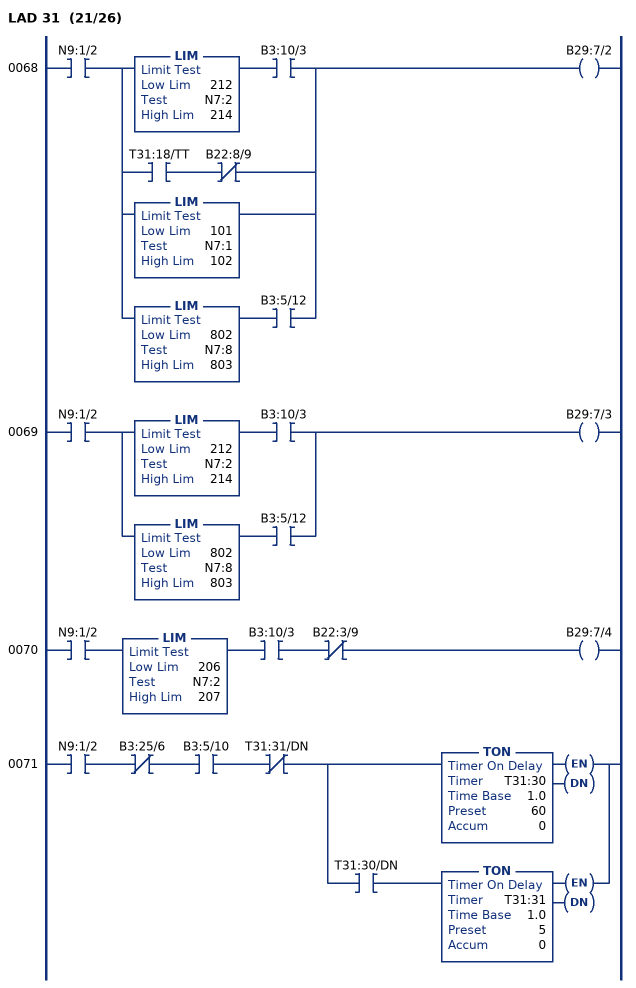
% Rung: 68 %
SOR XIC N9:1/2 BST LIM 212 N7:2 214 XIC B3:10/3 NXB XIC T31:18/TT XIO B22:8/9 NXB LIM 101 N7:1 102 NXB LIM 802 N7:8 803 XIC B3:5/12 BND OTE B29:7/2 EOR
% Rung: 69 %
SOR XIC N9:1/2 BST LIM 212 N7:2 214 XIC B3:10/3 NXB LIM 802 N7:8 803 XIC B3:5/12 BND OTE B29:7/3 EOR
% Rung: 70 %
SOR XIC N9:1/2 LIM 206 N7:2 207 XIC B3:10/3 XIO B22:3/9 OTE B29:7/4 EOR
% Rung: 71 %
SOR XIC N9:1/2 XIO B3:25/6 XIC B3:5/10 XIO T31:31/DN BST TON T31:30 1.0 60 0 NXB XIC T31:30/DN TON T31:31 1.0 5 0 BND EOR

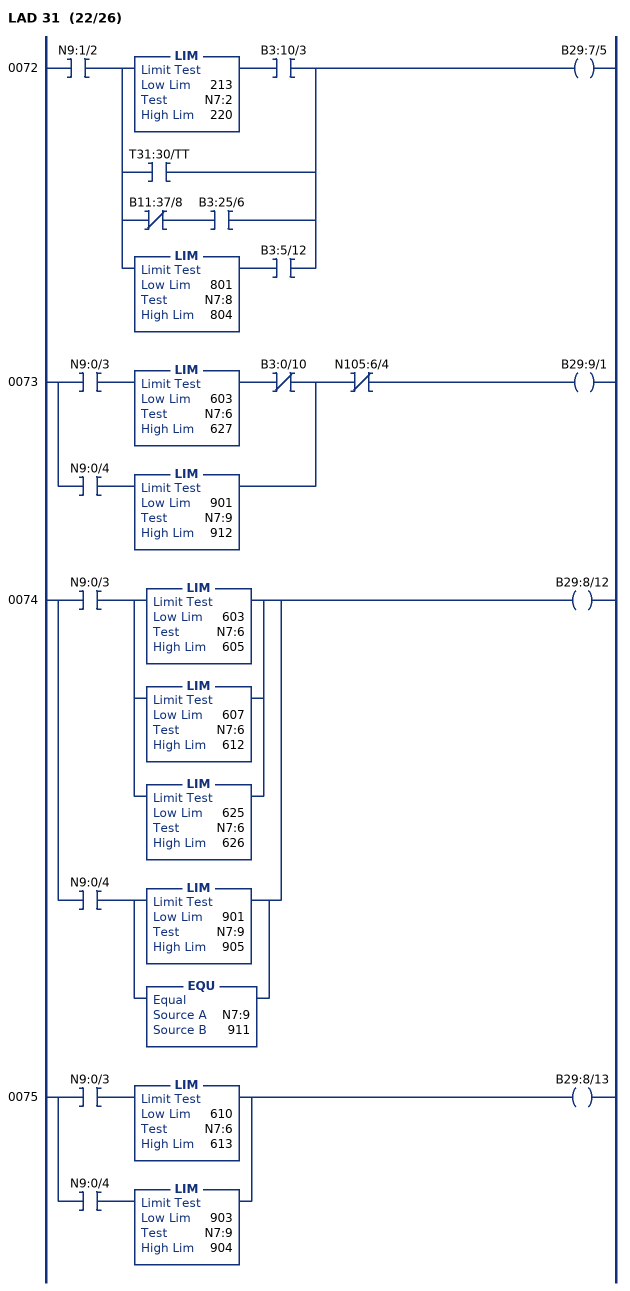
% Rung: 72 %
SOR XIC N9:1/2 BST LIM 213 N7:2 220 XIC B3:10/3 NXB XIC T31:30/TT NXB XIO B11:37/8 XIC B3:25/6 NXB LIM 801 N7:8 804 XIC B3:5/12 BND OTE B29:7/5 EOR
% Rung: 73 %
SOR BST XIC N9:0/3 LIM 603 N7:6 627 XIO B3:0/10 NXB XIC N9:0/4 LIM 901 N7:9 912 BND XIO N105:6/4 OTE B29:9/1 EOR
% Rung: 74 %
SOR BST XIC N9:0/3 BST LIM 603 N7:6 605 NXB LIM 607 N7:6 612 NXB LIM 625 N7:6 626 BND NXB XIC N9:0/4 BST LIM 901 N7:9 905 NXB EQU N7:9 911 BND BND OTE B29:8/12 EOR
% Rung: 75 %
SOR BST XIC N9:0/3 LIM 610 N7:6 613 NXB XIC N9:0/4 LIM 903 N7:9 904 BND OTE B29:8/13 EOR

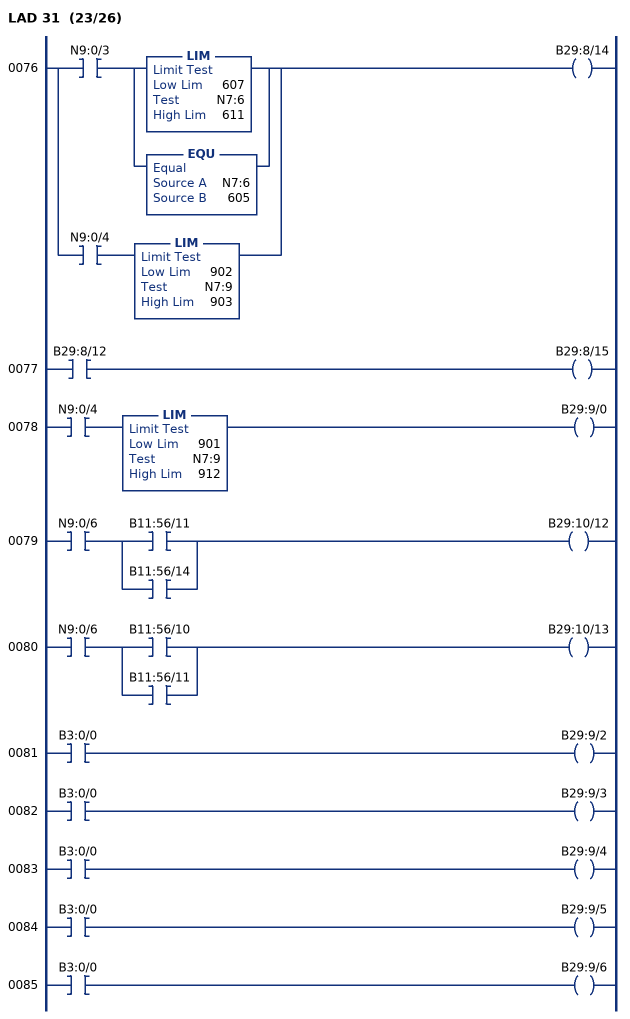
% Rung: 76 %
SOR BST XIC N9:0/3 BST LIM 607 N7:6 611 NXB EQU N7:6 605 BND NXB XIC N9:0/4 LIM 902 N7:9 903 BND OTE B29:8/14 EOR
% Rung: 77 %
SOR XIC B29:8/12 OTE B29:8/15 EOR
% Rung: 78 %
SOR XIC N9:0/4 LIM 901 N7:9 912 OTE B29:9/0 EOR
% Rung: 79 %
SOR XIC N9:0/6 BST XIC B11:56/11 NXB XIC B11:56/14 BND OTE B29:10/12 EOR
% Rung: 80 %
SOR XIC N9:0/6 BST XIC B11:56/10 NXB XIC B11:56/11 BND OTE B29:10/13 EOR
% Rung: 81 %
SOR XIC B3:0/0 OTE B29:9/2 EOR
% Rung: 82 %
SOR XIC B3:0/0 OTE B29:9/3 EOR
% Rung: 83 %
SOR XIC B3:0/0 OTE B29:9/4 EOR
% Rung: 84 %
SOR XIC B3:0/0 OTE B29:9/5 EOR
% Rung: 85 %
SOR XIC B3:0/0 OTE B29:9/6 EOR

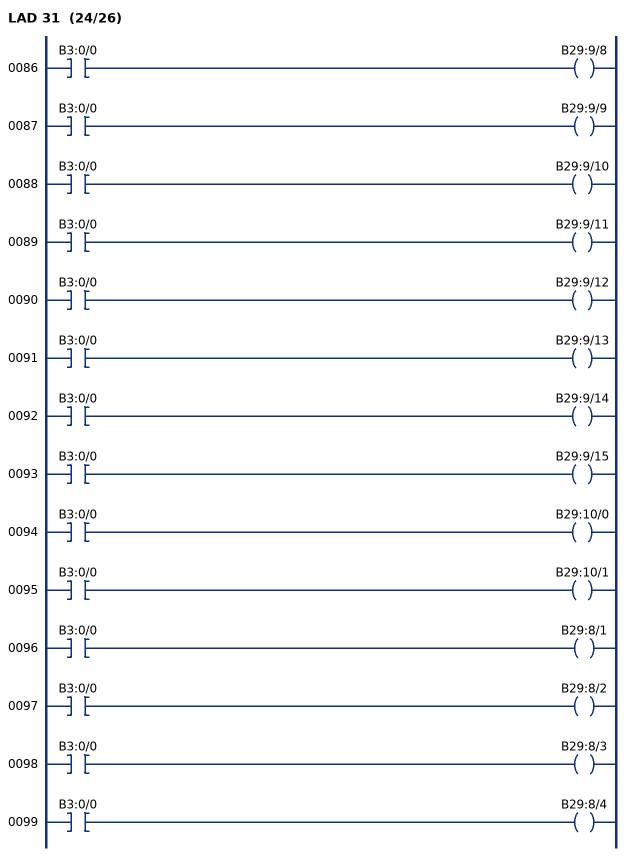
% Rung: 86 %
SOR XIC B3:0/0 OTE B29:9/8 EOR
% Rung: 87 %
SOR XIC B3:0/0 OTE B29:9/9 EOR
% Rung: 88 %
SOR XIC B3:0/0 OTE B29:9/10 EOR
% Rung: 89 %
SOR XIC B3:0/0 OTE B29:9/11 EOR
% Rung: 90 %
SOR XIC B3:0/0 OTE B29:9/12 EOR
% Rung: 91 %
SOR XIC B3:0/0 OTE B29:9/13 EOR
% Rung: 92 %
SOR XIC B3:0/0 OTE B29:9/14 EOR
% Rung: 93 %
SOR XIC B3:0/0 OTE B29:9/15 EOR
% Rung: 94 %
SOR XIC B3:0/0 OTE B29:10/0 EOR
% Rung: 95 %
SOR XIC B3:0/0 OTE B29:10/1 EOR
% Rung: 96 %
SOR XIC B3:0/0 OTE B29:8/1 EOR
% Rung: 97 %
SOR XIC B3:0/0 OTE B29:8/2 EOR
% Rung: 98 %
SOR XIC B3:0/0 OTE B29:8/3 EOR
% Rung: 99 %
SOR XIC B3:0/0 OTE B29:8/4 EOR

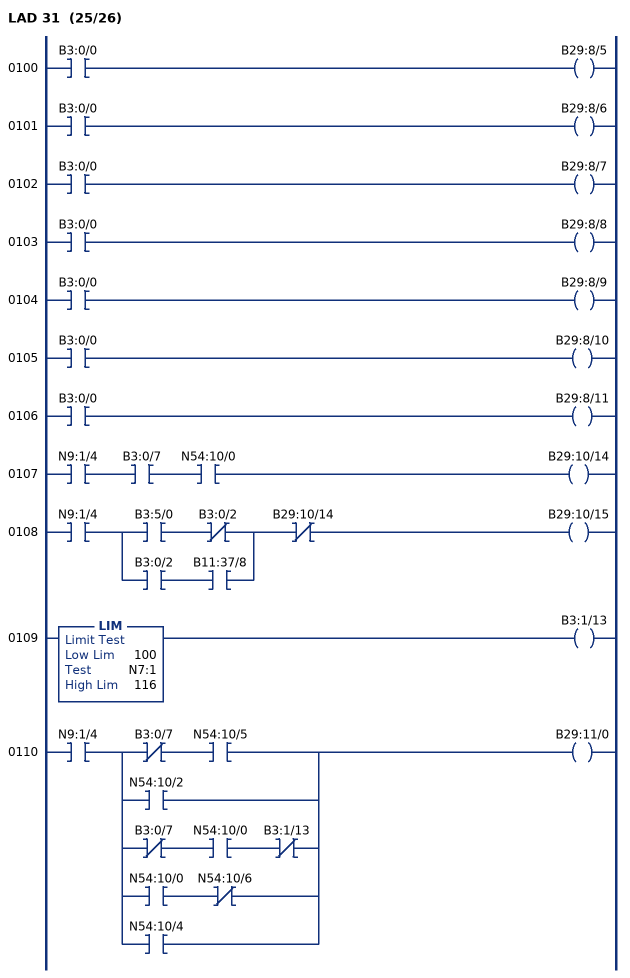
% Rung: 100 %
SOR XIC B3:0/0 OTE B29:8/5 EOR
% Rung: 101 %
SOR XIC B3:0/0 OTE B29:8/6 EOR
% Rung: 102 %
SOR XIC B3:0/0 OTE B29:8/7 EOR
% Rung: 103 %
SOR XIC B3:0/0 OTE B29:8/8 EOR
% Rung: 104 %
SOR XIC B3:0/0 OTE B29:8/9 EOR
% Rung: 105 %
SOR XIC B3:0/0 OTE B29:8/10 EOR
% Rung: 106 %
SOR XIC B3:0/0 OTE B29:8/11 EOR
% Rung: 107 %
SOR XIC N9:1/4 XIC B3:0/7 XIC N54:10/0 OTE B29:10/14 EOR
% Rung: 108 %
SOR XIC N9:1/4 BST XIC B3:5/0 XIO B3:0/2 NXB XIC B3:0/2 XIC B11:37/8 BND XIO B29:10/14 OTE B29:10/15 EOR
% Rung: 109 %
SOR LIM 100 N7:1 116 OTE B3:1/13 EOR
% Rung: 110 %
SOR XIC N9:1/4 BST XIO B3:0/7 XIC N54:10/5 NXB XIC N54:10/2 NXB XIO B3:0/7 XIC N54:10/0 XIO B3:1/13 NXB XIC N54:10/0 XIO N54:10/6 NXB XIC N54:10/4 BND OTE B29:11/0 EOR

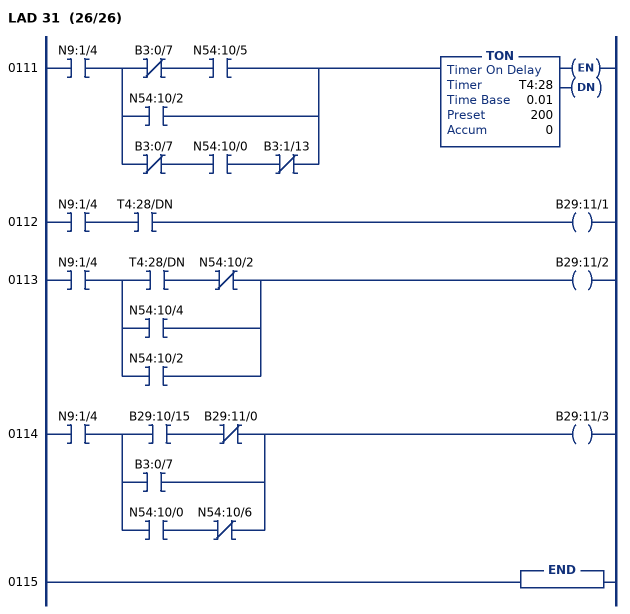
% Rung: 111 %
SOR XIC N9:1/4 BST XIO B3:0/7 XIC N54:10/5 NXB XIC N54:10/2 NXB XIO B3:0/7 XIC N54:10/0 XIO B3:1/13 BND TON T4:28 0.01 200 0 EOR
% Rung: 112 %
SOR XIC N9:1/4 XIC T4:28/DN OTE B29:11/1 EOR
% Rung: 113 %
SOR XIC N9:1/4 BST XIC T4:28/DN XIO N54:10/2 NXB XIC N54:10/4 NXB XIC N54:10/2 BND OTE B29:11/2 EOR
% Rung: 114 %
SOR XIC N9:1/4 BST XIC B29:10/15 XIO B29:11/0 NXB XIC B3:0/7 NXB XIC N54:10/0 XIO N54:10/6 BND OTE B29:11/3 EOR
% Rung: 115 %
SOR END EOR

LADDER 32
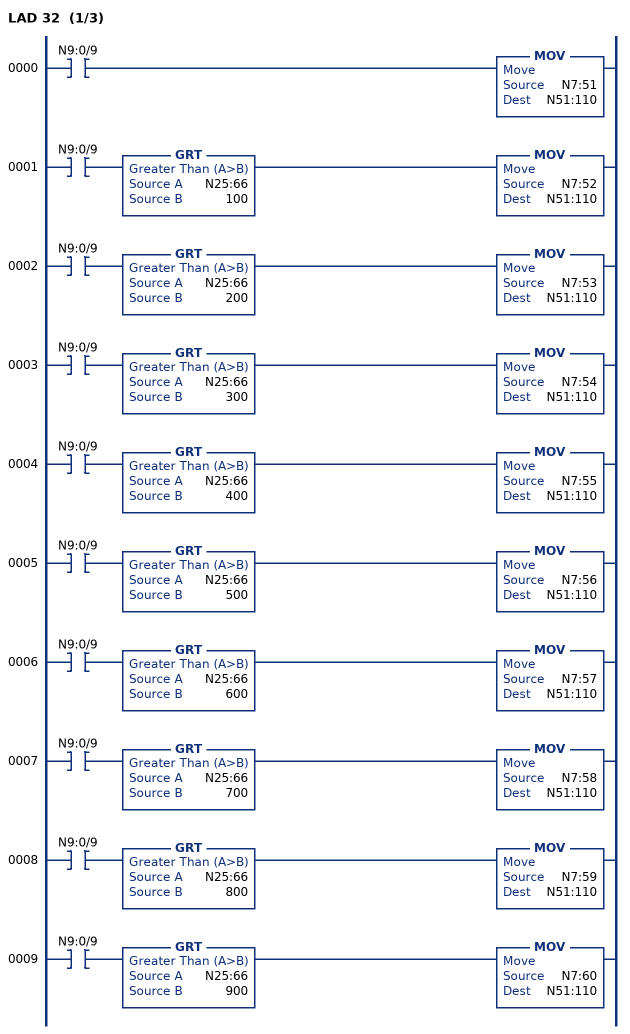
% Rung: 0 %
SOR XIC N9:0/9 MOV N7:51 N51:110 EOR
% Rung: 1 %
SOR XIC N9:0/9 GRT N25:66 100 MOV N7:52 N51:110 EOR
% Rung: 2 %
SOR XIC N9:0/9 GRT N25:66 200 MOV N7:53 N51:110 EOR
% Rung: 3 %
SOR XIC N9:0/9 GRT N25:66 300 MOV N7:54 N51:110 EOR
% Rung: 4 %
SOR XIC N9:0/9 GRT N25:66 400 MOV N7:55 N51:110 EOR
% Rung: 5 %
SOR XIC N9:0/9 GRT N25:66 500 MOV N7:56 N51:110 EOR
% Rung: 6 %
SOR XIC N9:0/9 GRT N25:66 600 MOV N7:57 N51:110 EOR
% Rung: 7 %
SOR XIC N9:0/9 GRT N25:66 700 MOV N7:58 N51:110 EOR
% Rung: 8 %
SOR XIC N9:0/9 GRT N25:66 800 MOV N7:59 N51:110 EOR
% Rung: 9 %
SOR XIC N9:0/9 GRT N25:66 900 MOV N7:60 N51:110 EOR

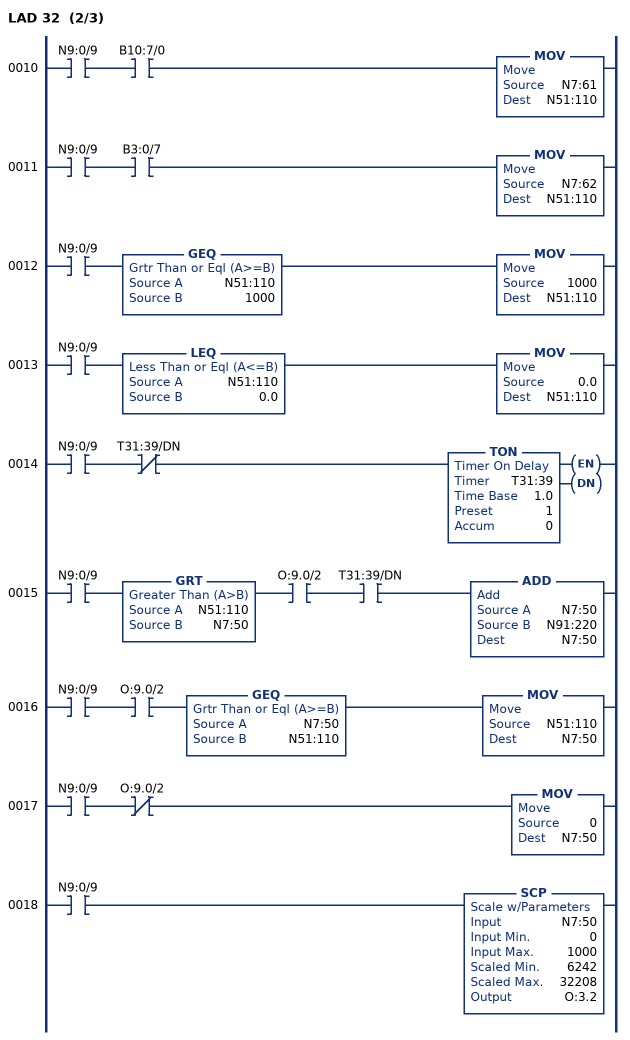
% Rung: 10 %
SOR XIC N9:0/9 XIC B10:7/0 MOV N7:61 N51:110 EOR
% Rung: 11 %
SOR XIC N9:0/9 XIC B3:0/7 MOV N7:62 N51:110 EOR
% Rung: 12 %
SOR XIC N9:0/9 GEQ N51:110 1000 MOV 1000 N51:110 EOR
% Rung: 13 %
SOR XIC N9:0/9 LEQ N51:110 0.0 MOV 0.0 N51:110 EOR
% Rung: 14 %
SOR XIC N9:0/9 XIO T31:39/DN TON T31:39 1.0 1 0 EOR
% Rung: 15 %
SOR XIC N9:0/9 GRT N51:110 N7:50 XIC O:9.0/2 XIC T31:39/DN ADD N7:50 N91:220 N7:50 EOR
% Rung: 16 %
SOR XIC N9:0/9 XIC O:9.0/2 GEQ N7:50 N51:110 MOV N51:110 N7:50 EOR
% Rung: 17 %
SOR XIC N9:0/9 XIO O:9.0/2 MOV 0 N7:50 EOR
% Rung: 18 %
SOR XIC N9:0/9 SCP N7:50 0 1000 6242 32208 O:3.2 EOR

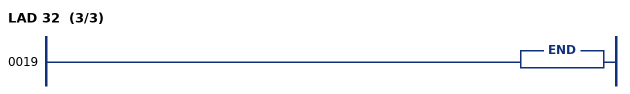
% Rung: 19 %
SOR END EOR

LADDER 40
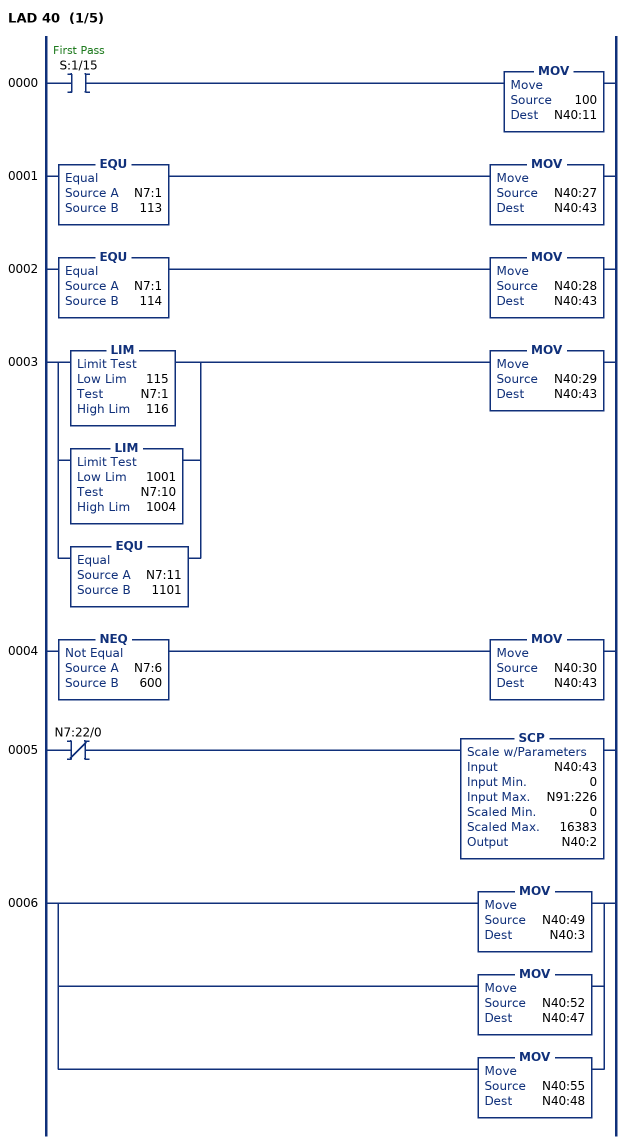
% Rung: 0 %
SOR XIC S:1/15 MOV 100 N40:11 EOR
%   S:1/15  "First Pass" %
% Rung: 1 %
SOR EQU N7:1 113 MOV N40:27 N40:43 EOR
% Rung: 2 %
SOR EQU N7:1 114 MOV N40:28 N40:43 EOR
% Rung: 3 %
SOR BST LIM 115 N7:1 116 NXB LIM 1001 N7:10 1004 NXB EQU N7:11 1101 BND MOV N40:29 N40:43 EOR
% Rung: 4 %
SOR NEQ N7:6 600 MOV N40:30 N40:43 EOR
% Rung: 5 %
SOR XIO N7:22/0 SCP N40:43 0 N91:226 0 16383 N40:2 EOR
% Rung: 6 %
SOR BST MOV N40:49 N40:3 NXB MOV N40:52 N40:47 NXB MOV N40:55 N40:48 BND EOR

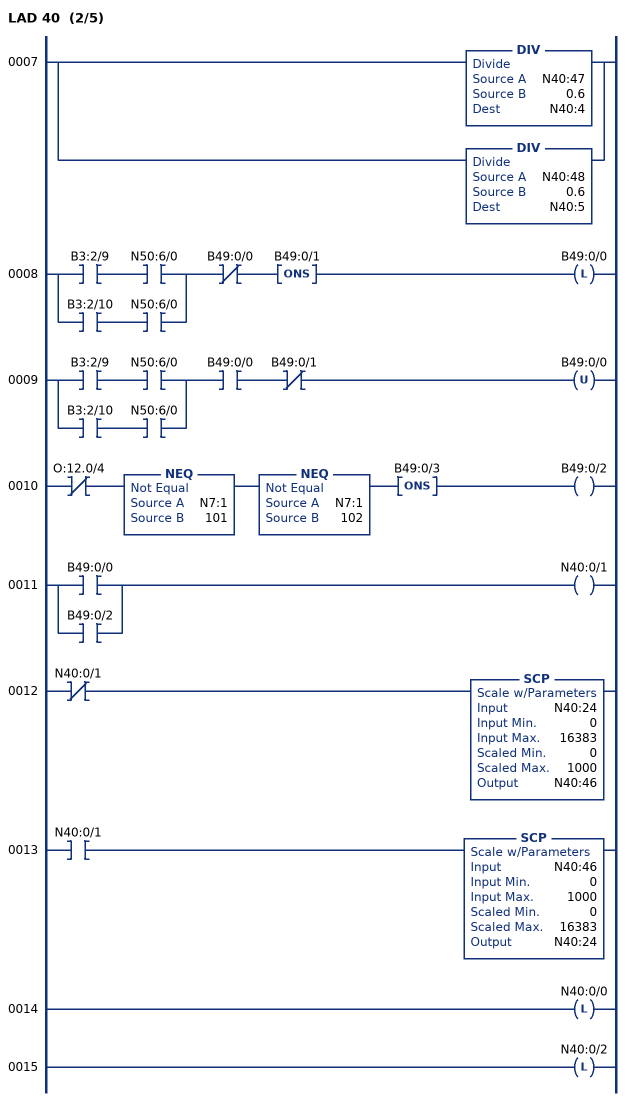
% Rung: 7 %
SOR BST DIV N40:47 0.6 N40:4 NXB DIV N40:48 0.6 N40:5 BND EOR
% Rung: 8 %
SOR BST XIC B3:2/9 XIC N50:6/0 NXB XIC B3:2/10 XIC N50:6/0 BND XIO B49:0/0 OSR B49:0/1 OTL B49:0/0 EOR
% Rung: 9 %
SOR BST XIC B3:2/9 XIC N50:6/0 NXB XIC B3:2/10 XIC N50:6/0 BND XIC B49:0/0 XIO B49:0/1 OTU B49:0/0 EOR
% Rung: 10 %
SOR XIO O:12.0/4 NEQ N7:1 101 NEQ N7:1 102 OSR B49:0/3 OTE B49:0/2 EOR
% Rung: 11 %
SOR BST XIC B49:0/0 NXB XIC B49:0/2 BND OTE N40:0/1 EOR
% Rung: 12 %
SOR XIO N40:0/1 SCP N40:24 0 16383 0 1000 N40:46 EOR
% Rung: 13 %
SOR XIC N40:0/1 SCP N40:46 0 1000 0 16383 N40:24 EOR
% Rung: 14 %
SOR OTL N40:0/0 EOR
% Rung: 15 %
SOR OTL N40:0/2 EOR

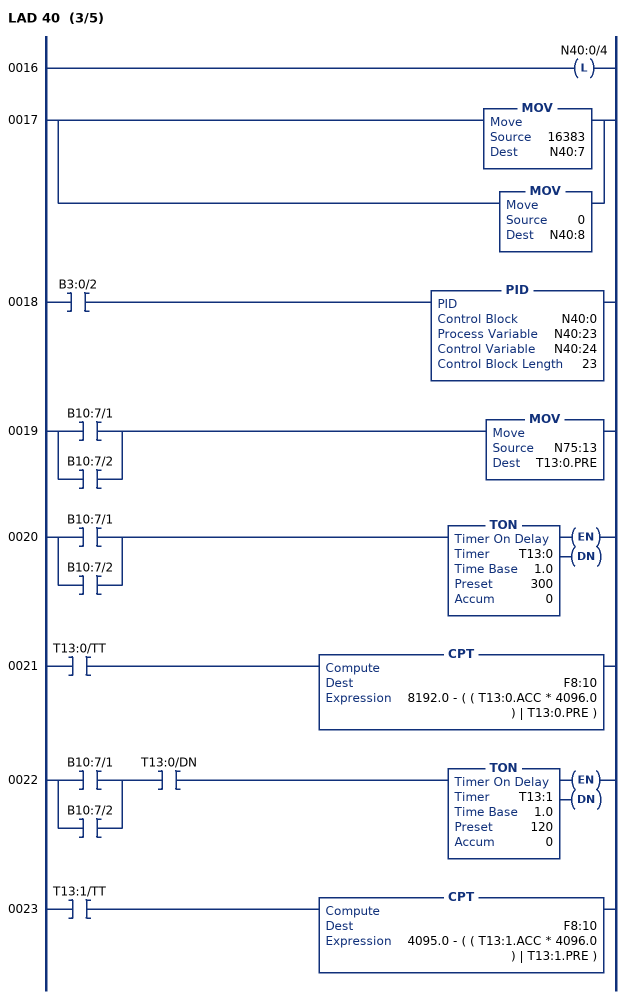
% Rung: 16 %
SOR OTL N40:0/4 EOR
% Rung: 17 %
SOR BST MOV 16383 N40:7 NXB MOV 0 N40:8 BND EOR
% Rung: 18 %
SOR XIC B3:0/2 PID N40:0 N40:23 N40:24 23 EOR
% Rung: 19 %
SOR BST XIC B10:7/1 NXB XIC B10:7/2 BND MOV N75:13 T13:0.PRE EOR
% Rung: 20 %
SOR BST XIC B10:7/1 NXB XIC B10:7/2 BND TON T13:0 1.0 300 0 EOR
% Rung: 21 %
SOR XIC T13:0/TT CPT F8:10 " 8192.0 - ( ( T13:0.ACC * 4096.0 ) | T13:0.PRE ) " EOR
% Rung: 22 %
SOR BST XIC B10:7/1 NXB XIC B10:7/2 BND XIC T13:0/DN TON T13:1 1.0 120 0 EOR
% Rung: 23 %
SOR XIC T13:1/TT CPT F8:10 " 4095.0 - ( ( T13:1.ACC * 4096.0 ) | T13:1.PRE ) " EOR

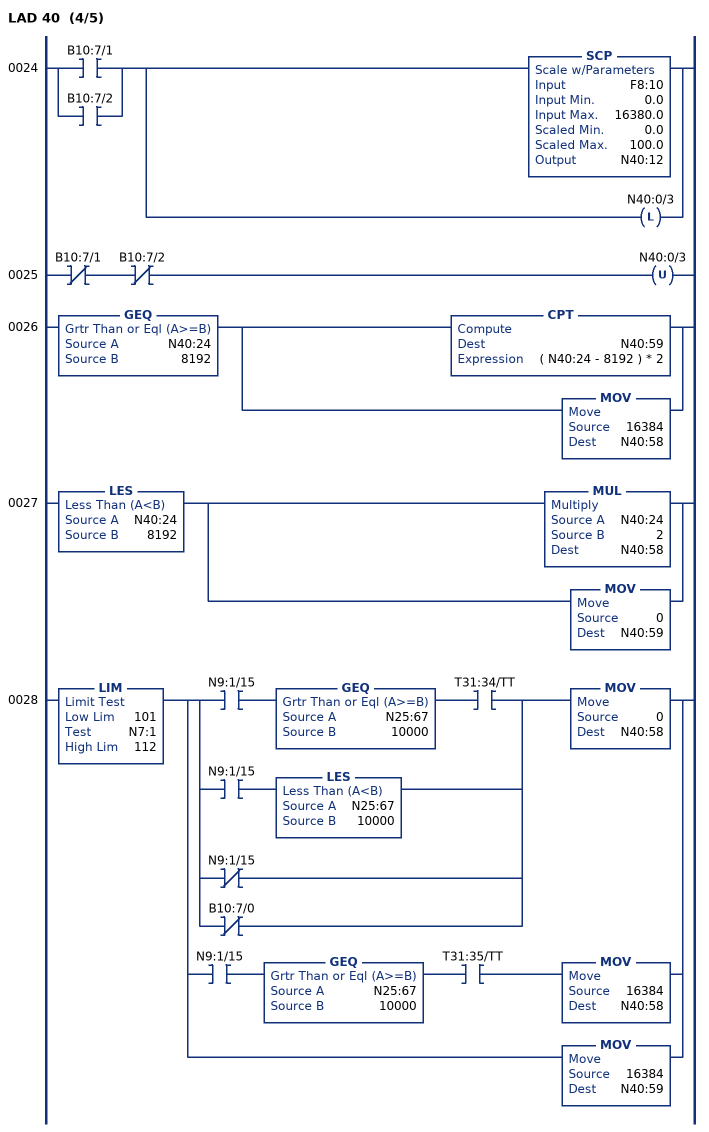
% Rung: 24 %
SOR BST XIC B10:7/1 NXB XIC B10:7/2 BND BST SCP F8:10 0.0 16380.0 0.0 100.0 N40:12 NXB OTL N40:0/3 BND EOR
% Rung: 25 %
SOR XIO B10:7/1 XIO B10:7/2 OTU N40:0/3 EOR
% Rung: 26 %
SOR GEQ N40:24 8192 BST CPT N40:59 " ( N40:24 - 8192 ) * 2 " NXB MOV 16384 N40:58 BND EOR
% Rung: 27 %
SOR LES N40:24 8192 BST MUL N40:24 2 N40:58 NXB MOV 0 N40:59 BND EOR
% Rung: 28 %
SOR LIM 101 N7:1 112 BST BST XIC N9:1/15 GEQ N25:67 10000 XIC T31:34/TT NXB XIC N9:1/15 LES N25:67 10000 NXB XIO N9:1/15 NXB XIO B10:7/0 BND MOV 0 N40:58 NXB XIC N9:1/15 GEQ N25:67 10000 XIC T31:35/TT MOV 16384 N40:58 NXB MOV 16384 N40:59 BND EOR

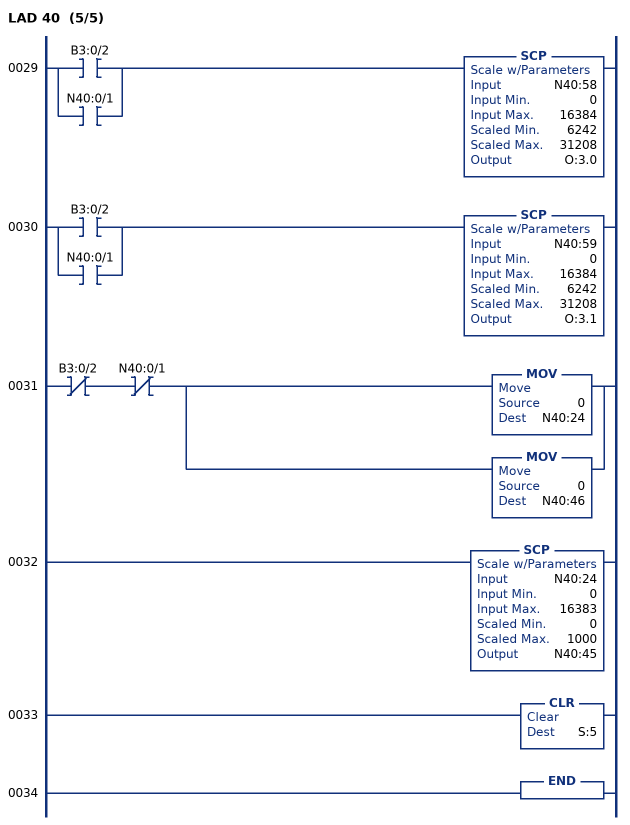
% Rung: 29 %
SOR BST XIC B3:0/2 NXB XIC N40:0/1 BND SCP N40:58 0 16384 6242 31208 O:3.0 EOR
% Rung: 30 %
SOR BST XIC B3:0/2 NXB XIC N40:0/1 BND SCP N40:59 0 16384 6242 31208 O:3.1 EOR
% Rung: 31 %
SOR XIO B3:0/2 XIO N40:0/1 BST MOV 0 N40:24 NXB MOV 0 N40:46 BND EOR
% Rung: 32 %
SOR SCP N40:24 0 16383 0 1000 N40:45 EOR
% Rung: 33 %
SOR CLR S:5 EOR
% Rung: 34 %
SOR END EOR

LADDER 50
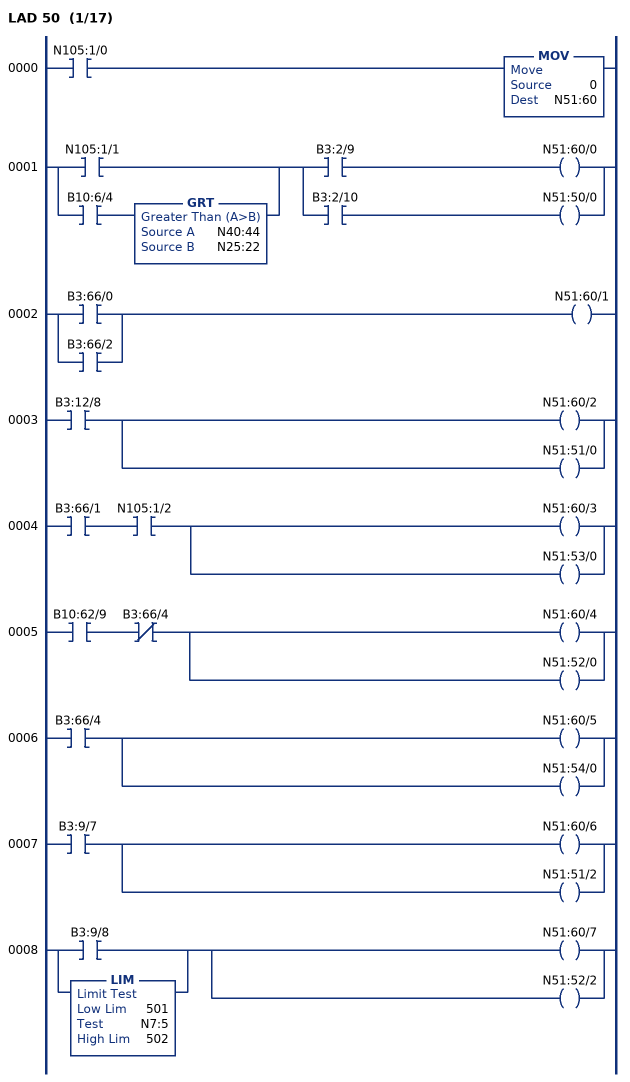
% Rung: 0 %
SOR XIC N105:1/0 MOV 0 N51:60 EOR
% Rung: 1 %
SOR BST XIC N105:1/1 NXB XIC B10:6/4 GRT N40:44 N25:22 BND BST XIC B3:2/9 OTE N51:60/0 NXB XIC B3:2/10 OTE N51:50/0 BND EOR
% Rung: 2 %
SOR BST XIC B3:66/0 NXB XIC B3:66/2 BND OTE N51:60/1 EOR
% Rung: 3 %
SOR XIC B3:12/8 BST OTE N51:60/2 NXB OTE N51:51/0 BND EOR
% Rung: 4 %
SOR XIC B3:66/1 XIC N105:1/2 BST OTE N51:60/3 NXB OTE N51:53/0 BND EOR
% Rung: 5 %
SOR XIC B10:62/9 XIO B3:66/4 BST OTE N51:60/4 NXB OTE N51:52/0 BND EOR
% Rung: 6 %
SOR XIC B3:66/4 BST OTE N51:60/5 NXB OTE N51:54/0 BND EOR
% Rung: 7 %
SOR XIC B3:9/7 BST OTE N51:60/6 NXB OTE N51:51/2 BND EOR
% Rung: 8 %
SOR BST XIC B3:9/8 NXB LIM 501 N7:5 502 BND BST OTE N51:60/7 NXB OTE N51:52/2 BND EOR

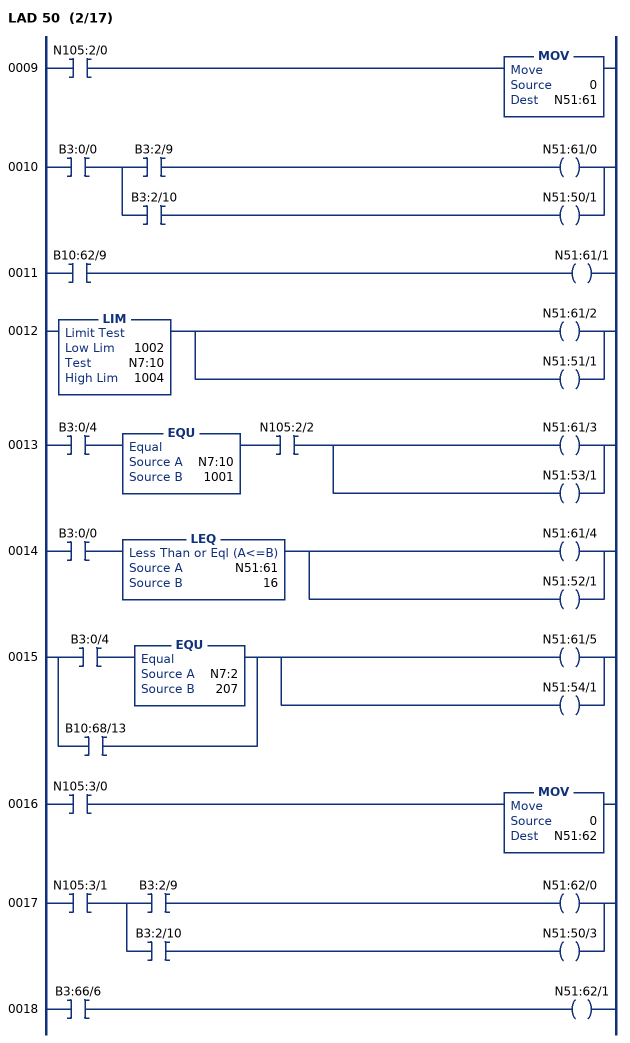
% Rung: 9 %
SOR XIC N105:2/0 MOV 0 N51:61 EOR
% Rung: 10 %
SOR XIC B3:0/0 BST XIC B3:2/9 OTE N51:61/0 NXB XIC B3:2/10 OTE N51:50/1 BND EOR
% Rung: 11 %
SOR XIC B10:62/9 OTE N51:61/1 EOR
% Rung: 12 %
SOR LIM 1002 N7:10 1004 BST OTE N51:61/2 NXB OTE N51:51/1 BND EOR
% Rung: 13 %
SOR XIC B3:0/4 EQU N7:10 1001 XIC N105:2/2 BST OTE N51:61/3 NXB OTE N51:53/1 BND EOR
% Rung: 14 %
SOR XIC B3:0/0 LEQ N51:61 16 BST OTE N51:61/4 NXB OTE N51:52/1 BND EOR
% Rung: 15 %
SOR BST XIC B3:0/4 EQU N7:2 207 NXB XIC B10:68/13 BND BST OTE N51:61/5 NXB OTE N51:54/1 BND EOR
% Rung: 16 %
SOR XIC N105:3/0 MOV 0 N51:62 EOR
% Rung: 17 %
SOR XIC N105:3/1 BST XIC B3:2/9 OTE N51:62/0 NXB XIC B3:2/10 OTE N51:50/3 BND EOR
% Rung: 18 %
SOR XIC B3:66/6 OTE N51:62/1 EOR

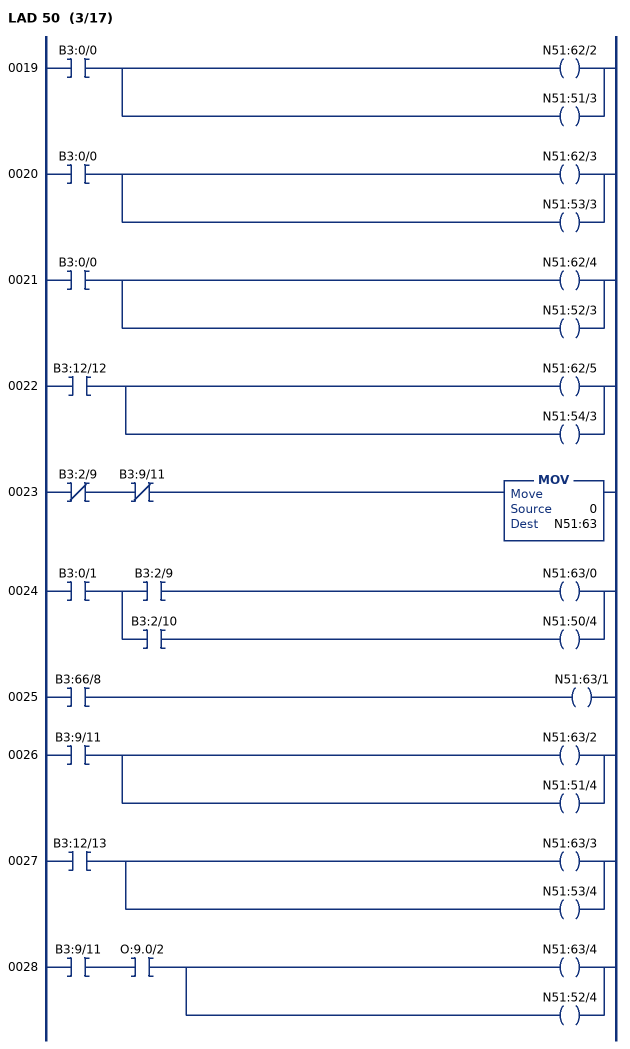
% Rung: 19 %
SOR XIC B3:0/0 BST OTE N51:62/2 NXB OTE N51:51/3 BND EOR
% Rung: 20 %
SOR XIC B3:0/0 BST OTE N51:62/3 NXB OTE N51:53/3 BND EOR
% Rung: 21 %
SOR XIC B3:0/0 BST OTE N51:62/4 NXB OTE N51:52/3 BND EOR
% Rung: 22 %
SOR XIC B3:12/12 BST OTE N51:62/5 NXB OTE N51:54/3 BND EOR
% Rung: 23 %
SOR XIO B3:2/9 XIO B3:9/11 MOV 0 N51:63 EOR
% Rung: 24 %
SOR XIC B3:0/1 BST XIC B3:2/9 OTE N51:63/0 NXB XIC B3:2/10 OTE N51:50/4 BND EOR
% Rung: 25 %
SOR XIC B3:66/8 OTE N51:63/1 EOR
% Rung: 26 %
SOR XIC B3:9/11 BST OTE N51:63/2 NXB OTE N51:51/4 BND EOR
% Rung: 27 %
SOR XIC B3:12/13 BST OTE N51:63/3 NXB OTE N51:53/4 BND EOR
% Rung: 28 %
SOR XIC B3:9/11 XIC O:9.0/2 BST OTE N51:63/4 NXB OTE N51:52/4 BND EOR

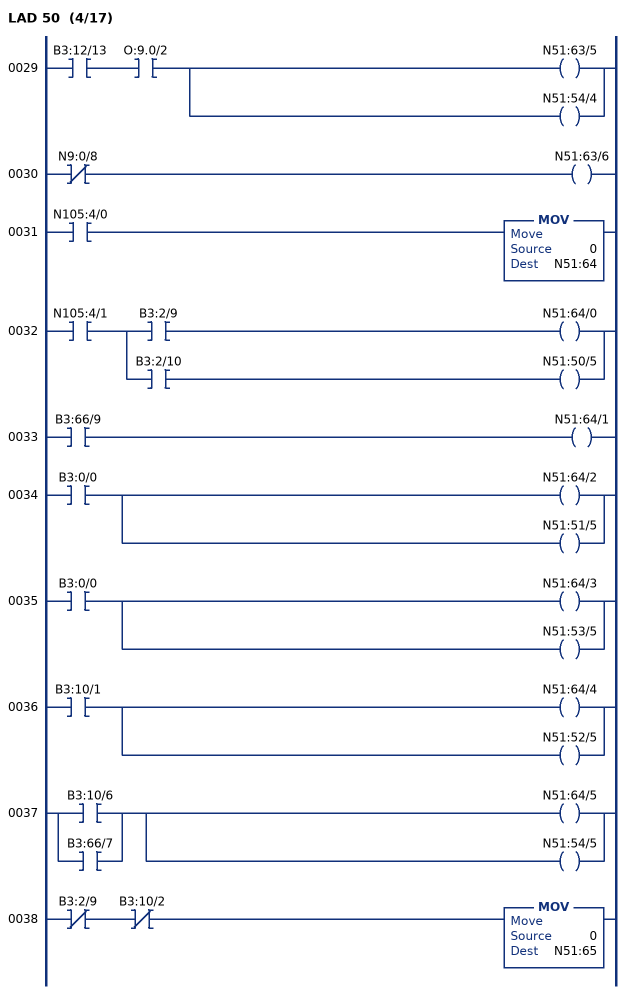
% Rung: 29 %
SOR XIC B3:12/13 XIC O:9.0/2 BST OTE N51:63/5 NXB OTE N51:54/4 BND EOR
% Rung: 30 %
SOR XIO N9:0/8 OTE N51:63/6 EOR
% Rung: 31 %
SOR XIC N105:4/0 MOV 0 N51:64 EOR
% Rung: 32 %
SOR XIC N105:4/1 BST XIC B3:2/9 OTE N51:64/0 NXB XIC B3:2/10 OTE N51:50/5 BND EOR
% Rung: 33 %
SOR XIC B3:66/9 OTE N51:64/1 EOR
% Rung: 34 %
SOR XIC B3:0/0 BST OTE N51:64/2 NXB OTE N51:51/5 BND EOR
% Rung: 35 %
SOR XIC B3:0/0 BST OTE N51:64/3 NXB OTE N51:53/5 BND EOR
% Rung: 36 %
SOR XIC B3:10/1 BST OTE N51:64/4 NXB OTE N51:52/5 BND EOR
% Rung: 37 %
SOR BST XIC B3:10/6 NXB XIC B3:66/7 BND BST OTE N51:64/5 NXB OTE N51:54/5 BND EOR
% Rung: 38 %
SOR XIO B3:2/9 XIO B3:10/2 MOV 0 N51:65 EOR

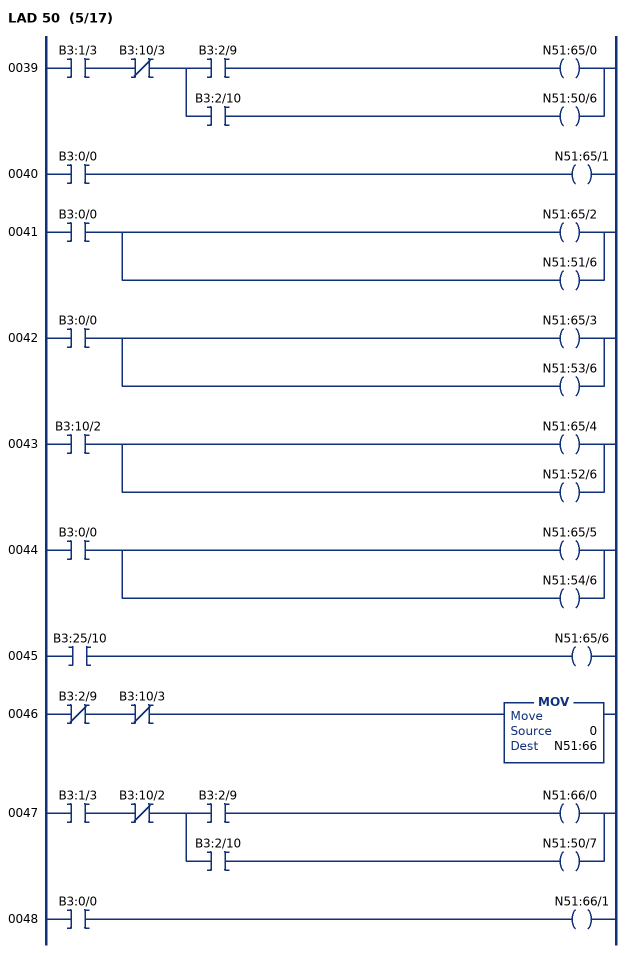
% Rung: 39 %
SOR XIC B3:1/3 XIO B3:10/3 BST XIC B3:2/9 OTE N51:65/0 NXB XIC B3:2/10 OTE N51:50/6 BND EOR
% Rung: 40 %
SOR XIC B3:0/0 OTE N51:65/1 EOR
% Rung: 41 %
SOR XIC B3:0/0 BST OTE N51:65/2 NXB OTE N51:51/6 BND EOR
% Rung: 42 %
SOR XIC B3:0/0 BST OTE N51:65/3 NXB OTE N51:53/6 BND EOR
% Rung: 43 %
SOR XIC B3:10/2 BST OTE N51:65/4 NXB OTE N51:52/6 BND EOR
% Rung: 44 %
SOR XIC B3:0/0 BST OTE N51:65/5 NXB OTE N51:54/6 BND EOR
% Rung: 45 %
SOR XIC B3:25/10 OTE N51:65/6 EOR
% Rung: 46 %
SOR XIO B3:2/9 XIO B3:10/3 MOV 0 N51:66 EOR
% Rung: 47 %
SOR XIC B3:1/3 XIO B3:10/2 BST XIC B3:2/9 OTE N51:66/0 NXB XIC B3:2/10 OTE N51:50/7 BND EOR
% Rung: 48 %
SOR XIC B3:0/0 OTE N51:66/1 EOR

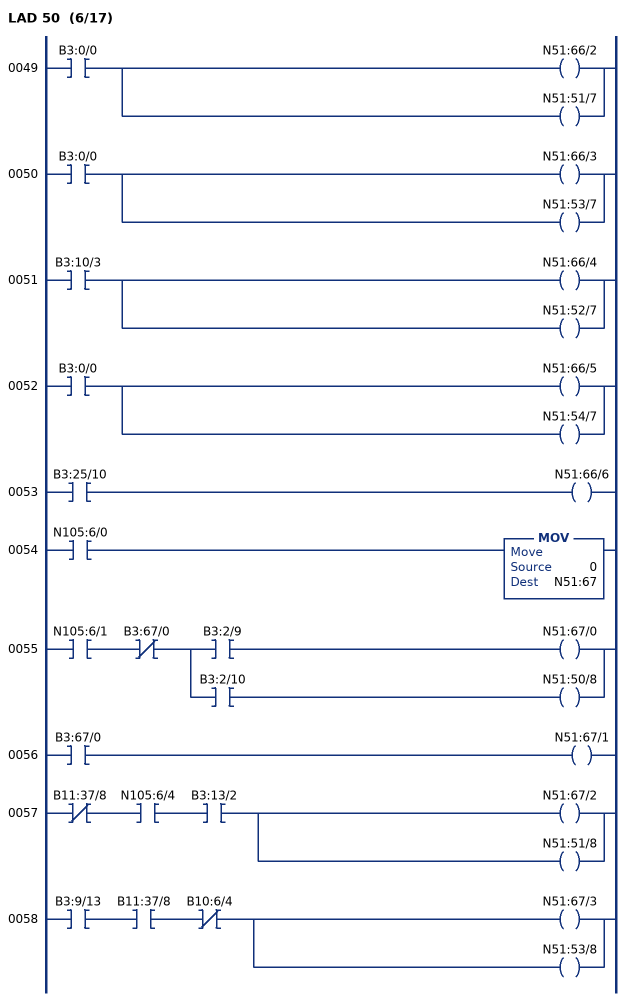
% Rung: 49 %
SOR XIC B3:0/0 BST OTE N51:66/2 NXB OTE N51:51/7 BND EOR
% Rung: 50 %
SOR XIC B3:0/0 BST OTE N51:66/3 NXB OTE N51:53/7 BND EOR
% Rung: 51 %
SOR XIC B3:10/3 BST OTE N51:66/4 NXB OTE N51:52/7 BND EOR
% Rung: 52 %
SOR XIC B3:0/0 BST OTE N51:66/5 NXB OTE N51:54/7 BND EOR
% Rung: 53 %
SOR XIC B3:25/10 OTE N51:66/6 EOR
% Rung: 54 %
SOR XIC N105:6/0 MOV 0 N51:67 EOR
% Rung: 55 %
SOR XIC N105:6/1 XIO B3:67/0 BST XIC B3:2/9 OTE N51:67/0 NXB XIC B3:2/10 OTE N51:50/8 BND EOR
% Rung: 56 %
SOR XIC B3:67/0 OTE N51:67/1 EOR
% Rung: 57 %
SOR XIO B11:37/8 XIC N105:6/4 XIC B3:13/2 BST OTE N51:67/2 NXB OTE N51:51/8 BND EOR
% Rung: 58 %
SOR XIC B3:9/13 XIC B11:37/8 XIO B10:6/4 BST OTE N51:67/3 NXB OTE N51:53/8 BND EOR

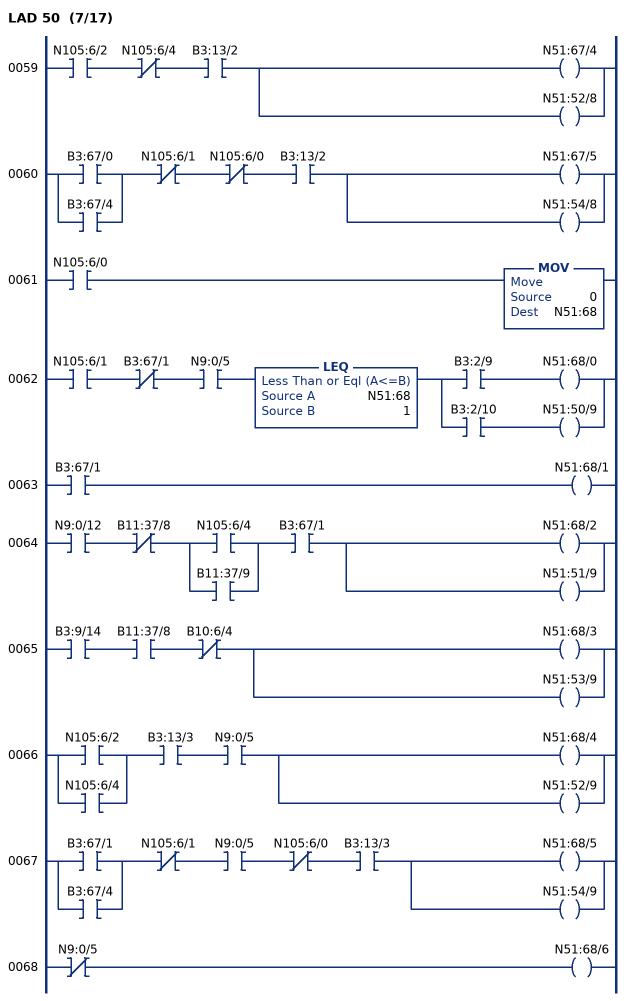
% Rung: 59 %
SOR XIC N105:6/2 XIO N105:6/4 XIC B3:13/2 BST OTE N51:67/4 NXB OTE N51:52/8 BND EOR
% Rung: 60 %
SOR BST XIC B3:67/0 NXB XIC B3:67/4 BND XIO N105:6/1 XIO N105:6/0 XIC B3:13/2 BST OTE N51:67/5 NXB OTE N51:54/8 BND EOR
% Rung: 61 %
SOR XIC N105:6/0 MOV 0 N51:68 EOR
% Rung: 62 %
SOR XIC N105:6/1 XIO B3:67/1 XIC N9:0/5 LEQ N51:68 1 BST XIC B3:2/9 OTE N51:68/0 NXB XIC B3:2/10 OTE N51:50/9 BND EOR
% Rung: 63 %
SOR XIC B3:67/1 OTE N51:68/1 EOR
% Rung: 64 %
SOR XIC N9:0/12 XIO B11:37/8 BST XIC N105:6/4 NXB XIC B11:37/9 BND XIC B3:67/1 BST OTE N51:68/2 NXB OTE N51:51/9 BND EOR
% Rung: 65 %
SOR XIC B3:9/14 XIC B11:37/8 XIO B10:6/4 BST OTE N51:68/3 NXB OTE N51:53/9 BND EOR
% Rung: 66 %
SOR BST XIC N105:6/2 NXB XIC N105:6/4 BND XIC B3:13/3 XIC N9:0/5 BST OTE N51:68/4 NXB OTE N51:52/9 BND EOR
% Rung: 67 %
SOR BST XIC B3:67/1 NXB XIC B3:67/4 BND XIO N105:6/1 XIC N9:0/5 XIO N105:6/0 XIC B3:13/3 BST OTE N51:68/5 NXB OTE N51:54/9 BND EOR
% Rung: 68 %
SOR XIO N9:0/5 OTE N51:68/6 EOR

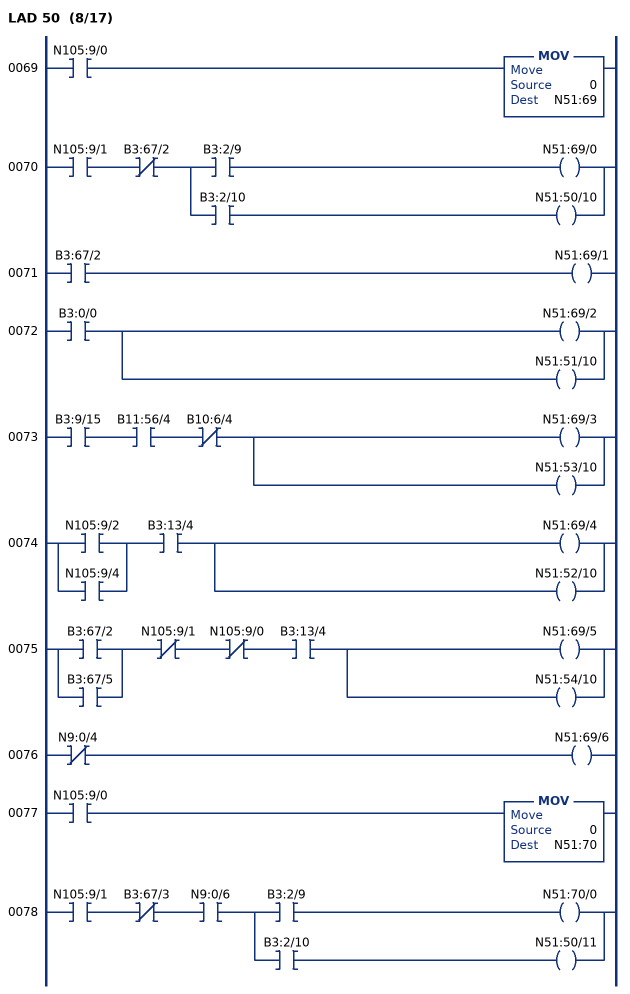
% Rung: 69 %
SOR XIC N105:9/0 MOV 0 N51:69 EOR
% Rung: 70 %
SOR XIC N105:9/1 XIO B3:67/2 BST XIC B3:2/9 OTE N51:69/0 NXB XIC B3:2/10 OTE N51:50/10 BND EOR
% Rung: 71 %
SOR XIC B3:67/2 OTE N51:69/1 EOR
% Rung: 72 %
SOR XIC B3:0/0 BST OTE N51:69/2 NXB OTE N51:51/10 BND EOR
% Rung: 73 %
SOR XIC B3:9/15 XIC B11:56/4 XIO B10:6/4 BST OTE N51:69/3 NXB OTE N51:53/10 BND EOR
% Rung: 74 %
SOR BST XIC N105:9/2 NXB XIC N105:9/4 BND XIC B3:13/4 BST OTE N51:69/4 NXB OTE N51:52/10 BND EOR
% Rung: 75 %
SOR BST XIC B3:67/2 NXB XIC B3:67/5 BND XIO N105:9/1 XIO N105:9/0 XIC B3:13/4 BST OTE N51:69/5 NXB OTE N51:54/10 BND EOR
% Rung: 76 %
SOR XIO N9:0/4 OTE N51:69/6 EOR
% Rung: 77 %
SOR XIC N105:9/0 MOV 0 N51:70 EOR
% Rung: 78 %
SOR XIC N105:9/1 XIO B3:67/3 XIC N9:0/6 BST XIC B3:2/9 OTE N51:70/0 NXB XIC B3:2/10 OTE N51:50/11 BND EOR

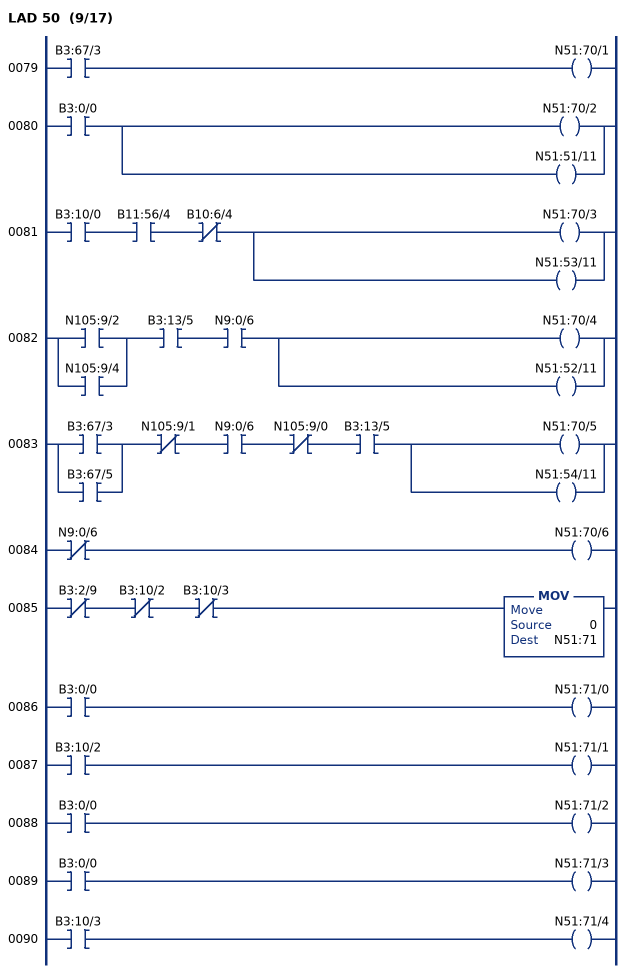
% Rung: 79 %
SOR XIC B3:67/3 OTE N51:70/1 EOR
% Rung: 80 %
SOR XIC B3:0/0 BST OTE N51:70/2 NXB OTE N51:51/11 BND EOR
% Rung: 81 %
SOR XIC B3:10/0 XIC B11:56/4 XIO B10:6/4 BST OTE N51:70/3 NXB OTE N51:53/11 BND EOR
% Rung: 82 %
SOR BST XIC N105:9/2 NXB XIC N105:9/4 BND XIC B3:13/5 XIC N9:0/6 BST OTE N51:70/4 NXB OTE N51:52/11 BND EOR
% Rung: 83 %
SOR BST XIC B3:67/3 NXB XIC B3:67/5 BND XIO N105:9/1 XIC N9:0/6 XIO N105:9/0 XIC B3:13/5 BST OTE N51:70/5 NXB OTE N51:54/11 BND EOR
% Rung: 84 %
SOR XIO N9:0/6 OTE N51:70/6 EOR
% Rung: 85 %
SOR XIO B3:2/9 XIO B3:10/2 XIO B3:10/3 MOV 0 N51:71 EOR
% Rung: 86 %
SOR XIC B3:0/0 OTE N51:71/0 EOR
% Rung: 87 %
SOR XIC B3:10/2 OTE N51:71/1 EOR
% Rung: 88 %
SOR XIC B3:0/0 OTE N51:71/2 EOR
% Rung: 89 %
SOR XIC B3:0/0 OTE N51:71/3 EOR
% Rung: 90 %
SOR XIC B3:10/3 OTE N51:71/4 EOR

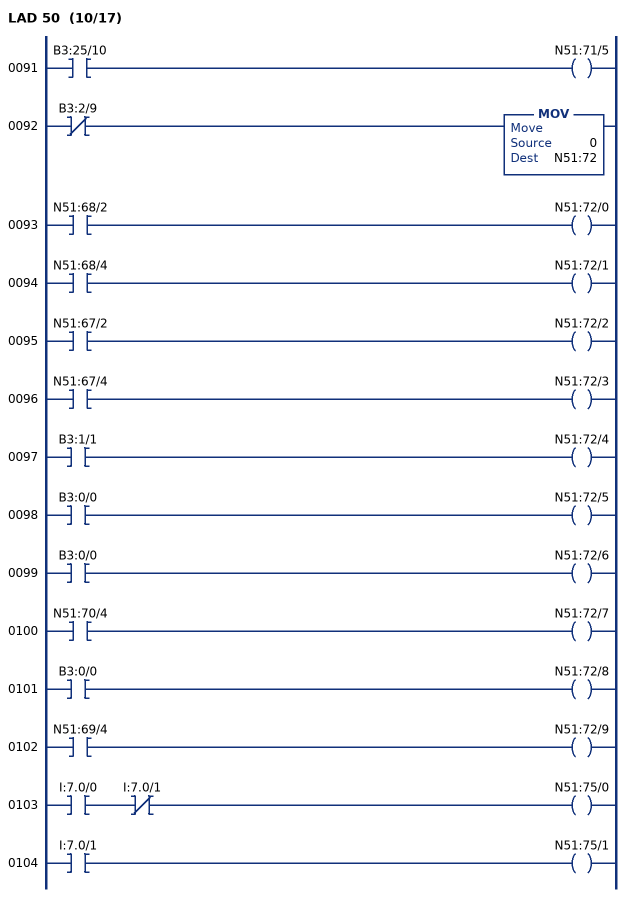
% Rung: 91 %
SOR XIC B3:25/10 OTE N51:71/5 EOR
% Rung: 92 %
SOR XIO B3:2/9 MOV 0 N51:72 EOR
% Rung: 93 %
SOR XIC N51:68/2 OTE N51:72/0 EOR
% Rung: 94 %
SOR XIC N51:68/4 OTE N51:72/1 EOR
% Rung: 95 %
SOR XIC N51:67/2 OTE N51:72/2 EOR
% Rung: 96 %
SOR XIC N51:67/4 OTE N51:72/3 EOR
% Rung: 97 %
SOR XIC B3:1/1 OTE N51:72/4 EOR
% Rung: 98 %
SOR XIC B3:0/0 OTE N51:72/5 EOR
% Rung: 99 %
SOR XIC B3:0/0 OTE N51:72/6 EOR
% Rung: 100 %
SOR XIC N51:70/4 OTE N51:72/7 EOR
% Rung: 101 %
SOR XIC B3:0/0 OTE N51:72/8 EOR
% Rung: 102 %
SOR XIC N51:69/4 OTE N51:72/9 EOR
% Rung: 103 %
SOR XIC I:7.0/0 XIO I:7.0/1 OTE N51:75/0 EOR
% Rung: 104 %
SOR XIC I:7.0/1 OTE N51:75/1 EOR

